Staubli VAL3: buildList2.pgx

program buildList2(num x_nViewMode)
  local num l_nSize
  local num i
  local string l_sName
  local bool l_bActive
  local num l_nValue
  local string l_sEmpty
  local string l_sField
  local string l_sItem
begin
  // INIT the list
  l_sEmpty=""
  call use:stringCopy(l_sEmpty,sList)
  // get the size
  call NUM:getSize(l_nSize)
  // Build the list
  for i=0 to l_nSize-1
    call NUM:get(l_sItem,i)
    call saveInOut:getItem_num(l_sName,l_sItem)
    call NUM:isActive(l_bActive,l_sItem)
    if l_bActive
      call saveInOut:getValue_num(l_nValue,l_sItem)
      // COUNTING
      call listAdd("["+toString("3",l_nValue)+"] "+l_sItem+" {"+l_sName+"}")
    endIf
  endFor
  // rebuild the list
  call use:listempty()
  call use:listadd(sList)
end
